Universal Robots PolyScope program: data_path_check_0p1s.urp

Program data_path_check_0p1s (installation=default directory=/programs/andyl createdIn=5.11.9.1010452 lastSavedIn=5.11.9.1010452 robotSerialNumber=20225200364)
Calibrated DH parameters: a=[0.00002, -0.569483, -0.54992, -0.00001, -0.000036, 0]; d=[0.180894, -146.691669, 192.918669, -46.053088, 0.119778, 0.115602]; alpha=[1.571425, -0.001534, 0.003359, 1.568739, -1.571477, 0]; deltaTheta=[0, 0.376258, -0.101074, -0.275185, -0.000002, 0]
Robot Program (runOnlyOnce=false)
  Script file /programs/andyl/demo-1.1/02_onrobot_data_path_check_wait_0p1s.script
    | def demo_1_1_write_onrobot_registers():
    |   write_output_float_register(24, Fx)
    |   write_output_float_register(25, Fy)
    |   write_output_float_register(26, Fz)
    |   write_output_float_register(27, Tx)
    |   write_output_float_register(28, Ty)
    |   write_output_float_register(29, Tz)
    | end
    | 
    | def demo_1_1_onrobot_data_path_check_wait_0p1s():
    |   cycles = 13
    |   i = 0
    | 
    |   textmsg("demo-1.1: OnRobot RTDE data path check 0.1s")
    |   while i < cycles:
    |     demo_1_1_write_onrobot_registers()
    |     sync()
    |     i = i + 1
    |   end
    |   demo_1_1_write_onrobot_registers()
    |   textmsg("demo-1.1: data path check finished")
    | end
    | 
    | demo_1_1_onrobot_data_path_check_wait_0p1s()
